TYPE TestLayoutStruct :
STRUCT
	_stackLayout: LayoutStackStruct;
	_uniformGridLayout: LayoutUniformGridStruct;
	_wrapLayout: LayoutWrapStruct;
	_tabsLayout: LayoutTabsStruct;
	_borderLayout: LayoutBorderStruct;
	_groupBoxLayout: LayoutGroupBoxStruct;
END_STRUCT
END_TYPE

(* stored: Version 1.1.0.1, ProductVersion 3.1.4024.9
   DUT TestLayoutStruct: Id {f29f5fcd-3df5-4eea-8c31-6186e4f5ace9} *)
